// TIA Portal V20 export
TYPE "s_PLC_Interlocks"
// stored: Access Published, IsFailsafeCompliant true, Namespace Safety
   STRUCT
      "Connection status" { ExternalWritable := 'False'; S7_SetPoint := 'True'} : "Safety.s_CONNECTION_STATUS";
      CellInterlocks { ExternalWritable := 'False'; S7_SetPoint := 'True'} : "Safety.s_zc_CellInterlocks";
      InterlockToAdjCellICSD { ExternalWritable := 'False'; S7_SetPoint := 'True'} : "Safety.s_zc_IntercellSafetyDeviceToAdjCell";
      NormalInterlocks { S7_SetPoint := 'True'} : "Safety.s_zc_NormalInterlocks";
      MiscInterlock { S7_SetPoint := 'True'} : "Safety.s_zc_MiscInterlocks";
   END_STRUCT;
END_TYPE
